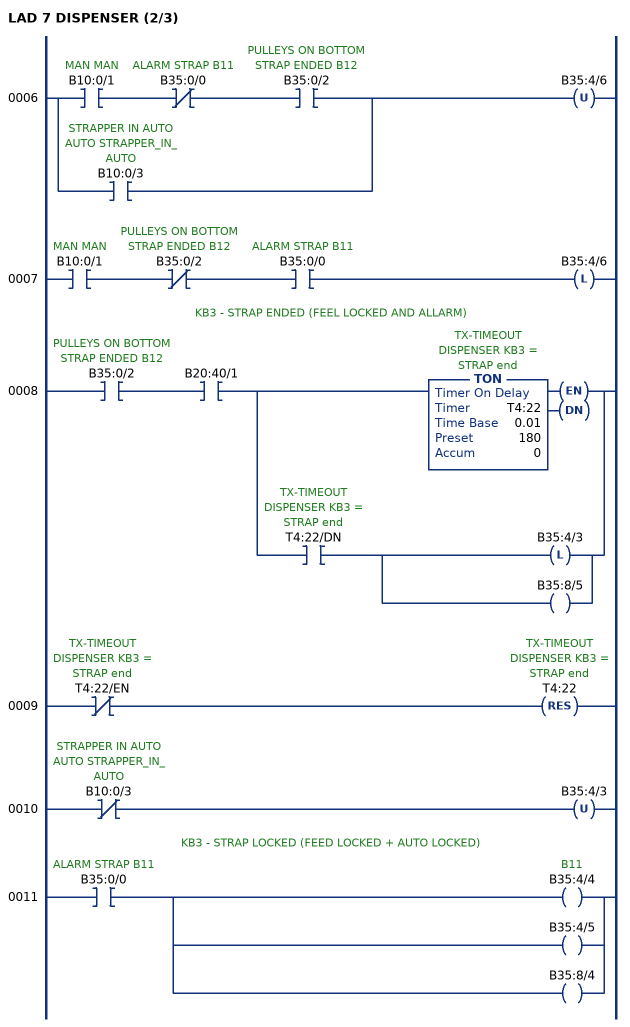
% Rung: 6 %
SOR BST XIC B10:0/1 XIO B35:0/0 XIC B35:0/2 NXB XIC B10:0/3 BND OTU B35:4/6 EOR
%   B10:0/1  MAN  "MAN" %
%   B35:0/0  B11  "ALARM STRAP" %
%   B35:0/2  B12  "PULLEYS ON BOTTOM STRAP ENDED" %
%   B10:0/3  STRAPPER_IN_AUTO  "STRAPPER IN AUTO AUTO" %
% Rung: 7 %
SOR XIC B10:0/1 XIO B35:0/2 XIC B35:0/0 OTL B35:4/6 EOR
%   B10:0/1  MAN  "MAN" %
%   B35:0/2  B12  "PULLEYS ON BOTTOM STRAP ENDED" %
%   B35:0/0  B11  "ALARM STRAP" %
% Rung: 8 %
% KB3 - STRAP ENDED (FEEL LOCKED AND ALLARM) %
SOR XIC B35:0/2 XIC B20:40/1 BST TON T4:22 0.01 180 0 NXB XIC T4:22/DN BST OTL B35:4/3 NXB OTE B35:8/5 BND BND EOR
%   B35:0/2  B12  "PULLEYS ON BOTTOM STRAP ENDED" %
%   T4:22  "TX-TIMEOUT DISPENSER KB3 = STRAP end" %
% Rung: 9 %
SOR XIO T4:22/EN RES T4:22 EOR
%   T4:22  "TX-TIMEOUT DISPENSER KB3 = STRAP end" %
% Rung: 10 %
SOR XIO B10:0/3 OTU B35:4/3 EOR
%   B10:0/3  STRAPPER_IN_AUTO  "STRAPPER IN AUTO AUTO" %
% Rung: 11 %
% KB3 - STRAP LOCKED (FEED LOCKED + AUTO LOCKED) %
SOR XIC B35:0/0 BST OTE B35:4/4 NXB BST OTE B35:4/5 NXB OTE B35:8/4 BND BND EOR
%   B35:0/0  B11  "ALARM STRAP" %
%   B35:4/4  "B11" %

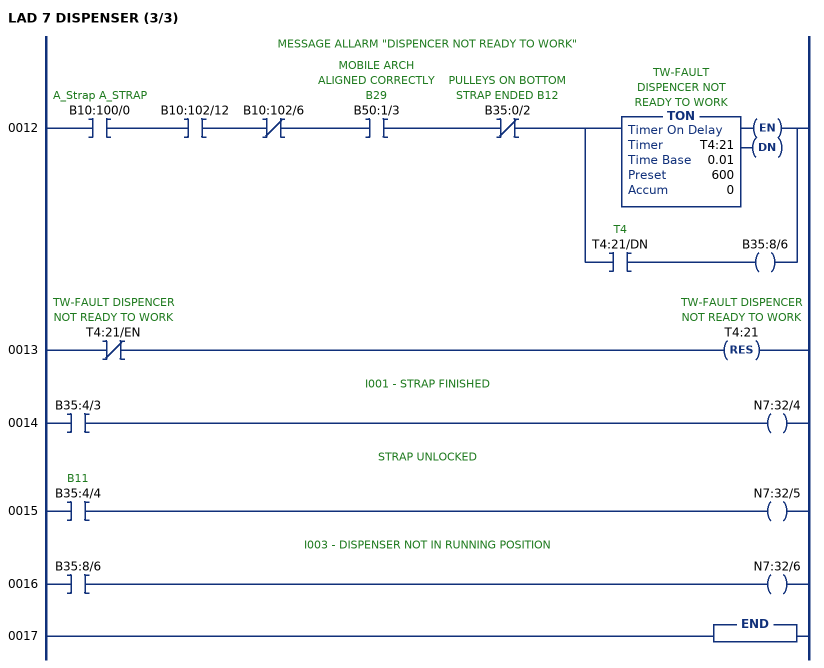
% Rung: 12 %
% MESSAGE ALLARM "DISPENCER NOT READY TO WORK" %
SOR XIC B10:100/0 XIC B10:102/12 XIO B10:102/6 XIC B50:1/3 XIO B35:0/2 BST TON T4:21 0.01 600 0 NXB XIC T4:21/DN OTE B35:8/6 BND EOR
%   B10:100/0  A_STRAP  "A_Strap" %
%   B50:1/3  B29  "MOBILE ARCH ALIGNED CORRECTLY" %
%   B35:0/2  B12  "PULLEYS ON BOTTOM STRAP ENDED" %
%   T4:21  "TW-FAULT DISPENCER NOT READY TO WORK" %
%   T4:21/DN  T4 %
% Rung: 13 %
SOR XIO T4:21/EN RES T4:21 EOR
%   T4:21  "TW-FAULT DISPENCER NOT READY TO WORK" %
% Rung: 14 %
% I001 - STRAP FINISHED %
SOR XIC B35:4/3 OTE N7:32/4 EOR
% Rung: 15 %
% STRAP UNLOCKED %
SOR XIC B35:4/4 OTE N7:32/5 EOR
%   B35:4/4  "B11" %
% Rung: 16 %
% I003 - DISPENSER NOT IN RUNNING POSITION %
SOR XIC B35:8/6 OTE N7:32/6 EOR
% Rung: 17 %
SOR END EOR

LADDER 8 "MH600"
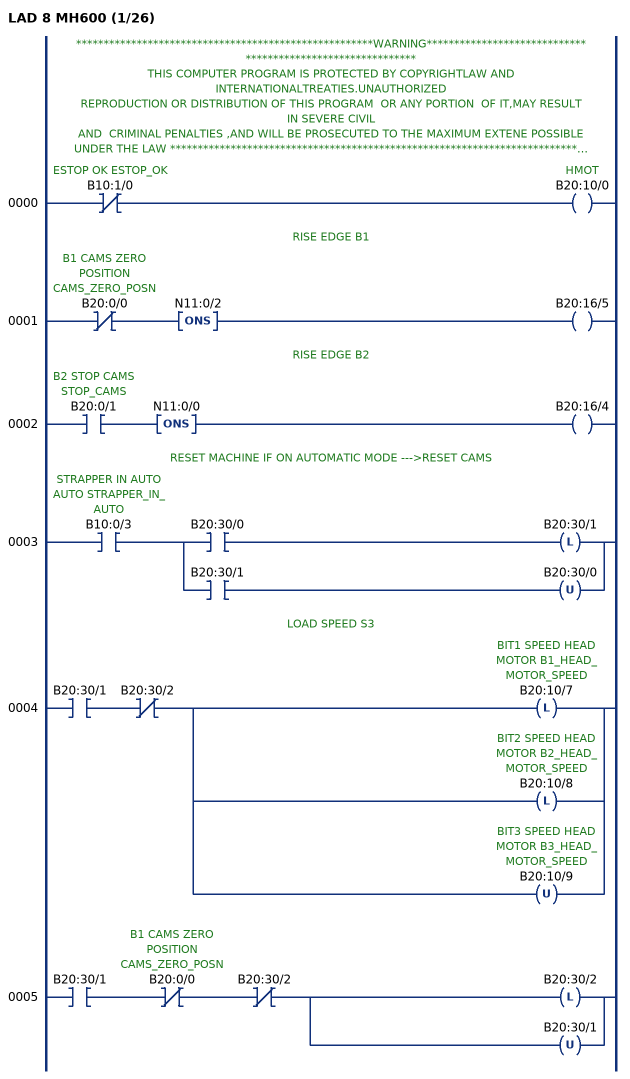
% Rung: 0 %
% ******************************************************WARNING************************************************************
% THIS COMPUTER PROGRAM IS PROTECTED BY COPYRIGHTLAW AND  INTERNATIONALTREATIES.UNAUTHORIZED
%  REPRODUCTION OR DISTRIBUTION OF THIS PROGRAM  OR ANY PORTION  OF IT,MAY RESULT IN SEVERE CIVIL
% AND  CRIMINAL PENALTIES ,AND WILL BE PROSECUTED TO THE MAXIMUM EXTENE POSSIBLE  UNDER THE LAW ************************************************************************************************************************** %
SOR XIO B10:1/0 OTE B20:10/0 EOR
%   B10:1/0  ESTOP_OK  "ESTOP OK" %
%   B20:10/0  "HMOT" %
% Rung: 1 %
% RISE EDGE B1 %
SOR XIO B20:0/0 ONS N11:0/2 OTE B20:16/5 EOR
%   B20:0/0  CAMS_ZERO_POSN  "B1 CAMS ZERO POSITION" %
% Rung: 2 %
% RISE EDGE B2 %
SOR XIC B20:0/1 ONS N11:0/0 OTE B20:16/4 EOR
%   B20:0/1  STOP_CAMS  "B2 STOP CAMS" %
% Rung: 3 %
% RESET MACHINE IF ON AUTOMATIC MODE --->RESET CAMS %
SOR XIC B10:0/3 BST XIC B20:30/0 OTL B20:30/1 NXB XIC B20:30/1 OTU B20:30/0 BND EOR
%   B10:0/3  STRAPPER_IN_AUTO  "STRAPPER IN AUTO AUTO" %
% Rung: 4 %
% LOAD SPEED S3 %
SOR XIC B20:30/1 XIO B20:30/2 BST OTL B20:10/7 NXB BST OTL B20:10/8 NXB OTU B20:10/9 BND BND EOR
%   B20:10/7  B1_HEAD_MOTOR_SPEED  "BIT1 SPEED HEAD MOTOR" %
%   B20:10/8  B2_HEAD_MOTOR_SPEED  "BIT2 SPEED HEAD MOTOR" %
%   B20:10/9  B3_HEAD_MOTOR_SPEED  "BIT3 SPEED HEAD MOTOR" %
% Rung: 5 %
SOR XIC B20:30/1 XIO B20:0/0 XIO B20:30/2 BST OTL B20:30/2 NXB OTU B20:30/1 BND EOR
%   B20:0/0  CAMS_ZERO_POSN  "B1 CAMS ZERO POSITION" %

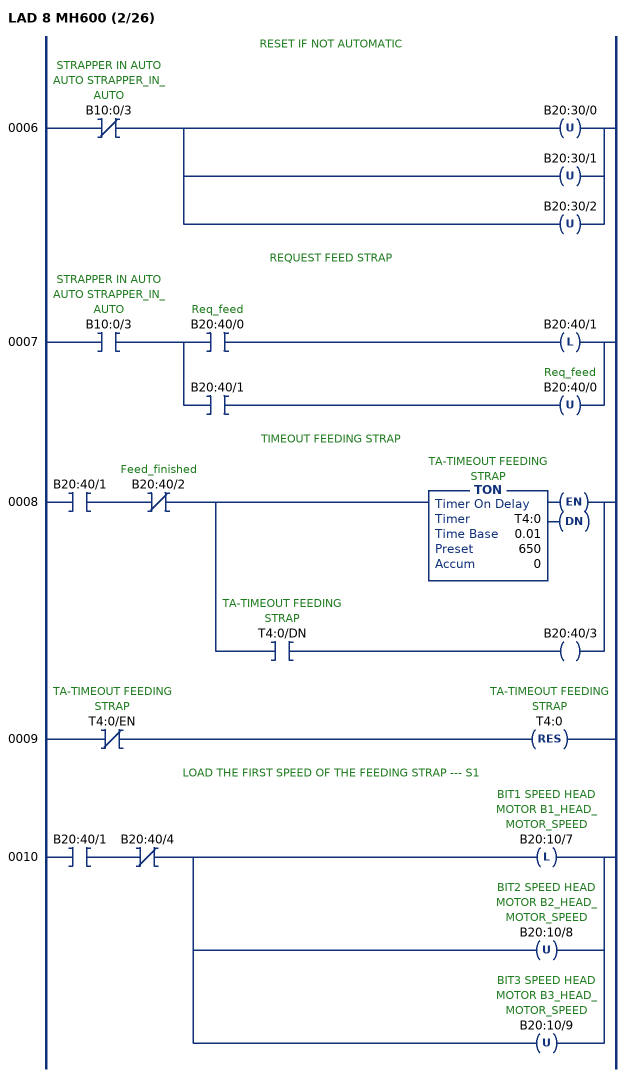
% Rung: 6 %
% RESET IF NOT AUTOMATIC %
SOR XIO B10:0/3 BST OTU B20:30/0 NXB BST OTU B20:30/1 NXB OTU B20:30/2 BND BND EOR
%   B10:0/3  STRAPPER_IN_AUTO  "STRAPPER IN AUTO AUTO" %
% Rung: 7 %
% REQUEST FEED STRAP %
SOR XIC B10:0/3 BST XIC B20:40/0 OTL B20:40/1 NXB XIC B20:40/1 OTU B20:40/0 BND EOR
%   B10:0/3  STRAPPER_IN_AUTO  "STRAPPER IN AUTO AUTO" %
%   B20:40/0  "Req_feed" %
% Rung: 8 %
% TIMEOUT FEEDING STRAP %
SOR XIC B20:40/1 XIO B20:40/2 BST TON T4:0 0.01 650 0 NXB XIC T4:0/DN OTE B20:40/3 BND EOR
%   B20:40/2  "Feed_finished" %
%   T4:0  "TA-TIMEOUT FEEDING STRAP" %
% Rung: 9 %
SOR XIO T4:0/EN RES T4:0 EOR
%   T4:0  "TA-TIMEOUT FEEDING STRAP" %
% Rung: 10 %
% LOAD THE FIRST SPEED OF THE FEEDING STRAP --- S1 %
SOR XIC B20:40/1 XIO B20:40/4 BST OTL B20:10/7 NXB BST OTU B20:10/8 NXB OTU B20:10/9 BND BND EOR
%   B20:10/7  B1_HEAD_MOTOR_SPEED  "BIT1 SPEED HEAD MOTOR" %
%   B20:10/8  B2_HEAD_MOTOR_SPEED  "BIT2 SPEED HEAD MOTOR" %
%   B20:10/9  B3_HEAD_MOTOR_SPEED  "BIT3 SPEED HEAD MOTOR" %

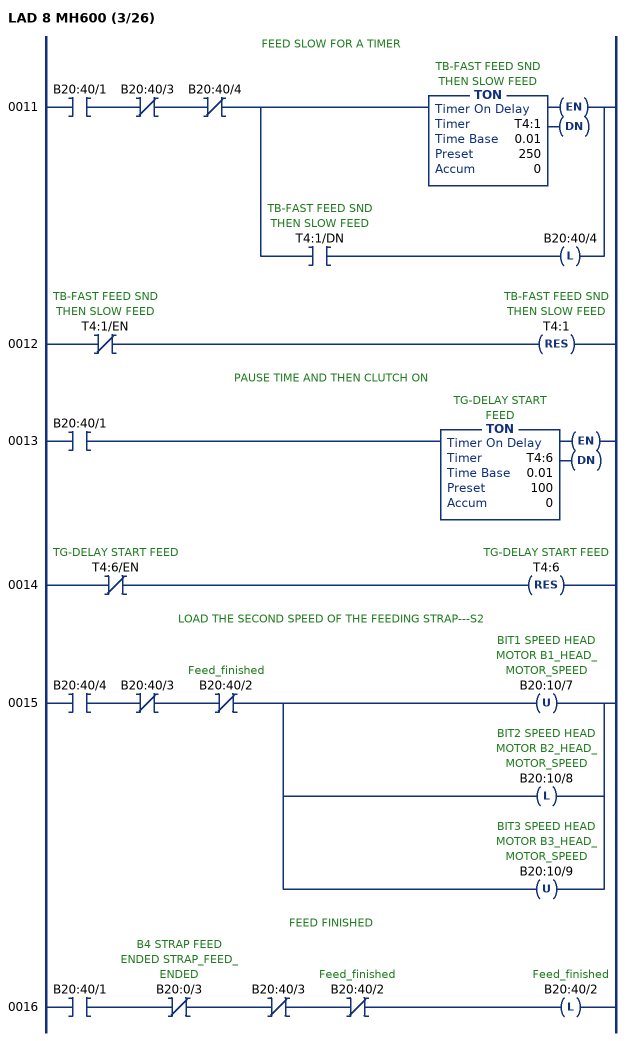
% Rung: 11 %
% FEED SLOW FOR A TIMER %
SOR XIC B20:40/1 XIO B20:40/3 XIO B20:40/4 BST TON T4:1 0.01 250 0 NXB XIC T4:1/DN OTL B20:40/4 BND EOR
%   T4:1  "TB-FAST FEED SND THEN SLOW FEED" %
% Rung: 12 %
SOR XIO T4:1/EN RES T4:1 EOR
%   T4:1  "TB-FAST FEED SND THEN SLOW FEED" %
% Rung: 13 %
% PAUSE TIME AND THEN CLUTCH ON %
SOR XIC B20:40/1 TON T4:6 0.01 100 0 EOR
%   T4:6  "TG-DELAY START FEED" %
% Rung: 14 %
SOR XIO T4:6/EN RES T4:6 EOR
%   T4:6  "TG-DELAY START FEED" %
% Rung: 15 %
% LOAD THE SECOND SPEED OF THE FEEDING STRAP---S2 %
SOR XIC B20:40/4 XIO B20:40/3 XIO B20:40/2 BST OTU B20:10/7 NXB BST OTL B20:10/8 NXB OTU B20:10/9 BND BND EOR
%   B20:40/2  "Feed_finished" %
%   B20:10/7  B1_HEAD_MOTOR_SPEED  "BIT1 SPEED HEAD MOTOR" %
%   B20:10/8  B2_HEAD_MOTOR_SPEED  "BIT2 SPEED HEAD MOTOR" %
%   B20:10/9  B3_HEAD_MOTOR_SPEED  "BIT3 SPEED HEAD MOTOR" %
% Rung: 16 %
% FEED FINISHED %
SOR XIC B20:40/1 XIO B20:0/3 XIO B20:40/3 XIO B20:40/2 OTL B20:40/2 EOR
%   B20:0/3  STRAP_FEED_ENDED  "B4 STRAP FEED ENDED" %
%   B20:40/2  "Feed_finished" %

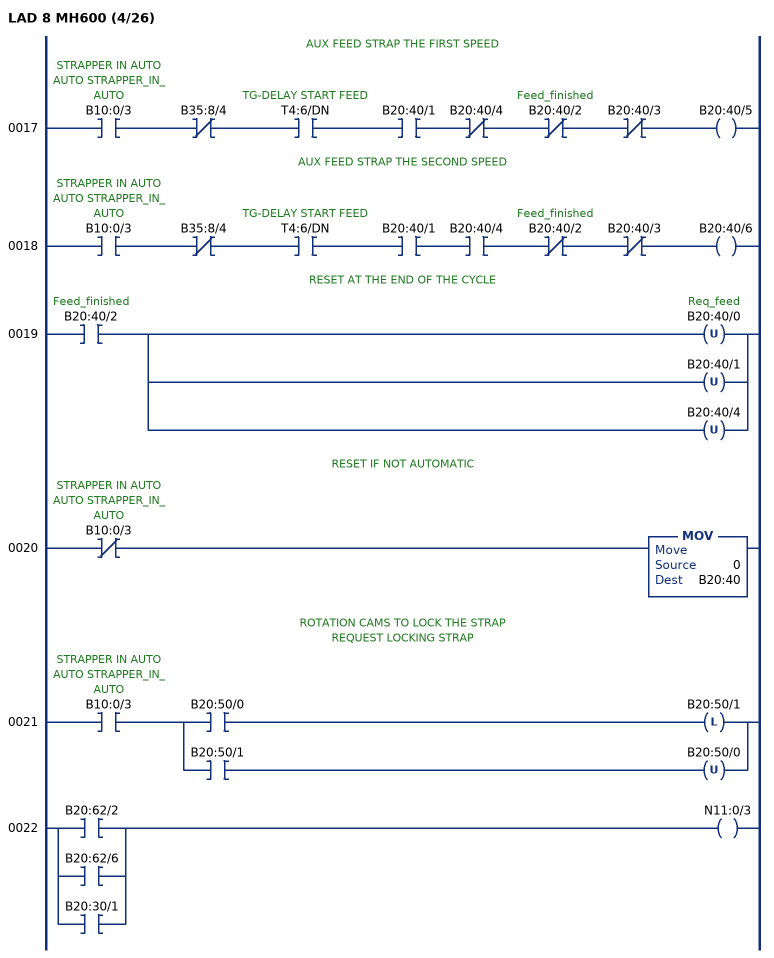
% Rung: 17 %
% AUX FEED STRAP THE FIRST SPEED %
SOR XIC B10:0/3 XIO B35:8/4 XIC T4:6/DN XIC B20:40/1 XIO B20:40/4 XIO B20:40/2 XIO B20:40/3 OTE B20:40/5 EOR
%   B10:0/3  STRAPPER_IN_AUTO  "STRAPPER IN AUTO AUTO" %
%   T4:6  "TG-DELAY START FEED" %
%   B20:40/2  "Feed_finished" %
% Rung: 18 %
% AUX FEED STRAP THE SECOND SPEED %
SOR XIC B10:0/3 XIO B35:8/4 XIC T4:6/DN XIC B20:40/1 XIC B20:40/4 XIO B20:40/2 XIO B20:40/3 OTE B20:40/6 EOR
%   B10:0/3  STRAPPER_IN_AUTO  "STRAPPER IN AUTO AUTO" %
%   T4:6  "TG-DELAY START FEED" %
%   B20:40/2  "Feed_finished" %
% Rung: 19 %
% RESET AT THE END OF THE CYCLE %
SOR XIC B20:40/2 BST OTU B20:40/0 NXB BST OTU B20:40/1 NXB OTU B20:40/4 BND BND EOR
%   B20:40/2  "Feed_finished" %
%   B20:40/0  "Req_feed" %
% Rung: 20 %
% RESET IF NOT AUTOMATIC %
SOR XIO B10:0/3 MOV 0 B20:40 EOR
%   B10:0/3  STRAPPER_IN_AUTO  "STRAPPER IN AUTO AUTO" %
% Rung: 21 %
% ROTATION CAMS TO LOCK THE STRAP
% REQUEST LOCKING STRAP %
SOR XIC B10:0/3 BST XIC B20:50/0 OTL B20:50/1 NXB XIC B20:50/1 OTU B20:50/0 BND EOR
%   B10:0/3  STRAPPER_IN_AUTO  "STRAPPER IN AUTO AUTO" %
% Rung: 22 %
SOR BST XIC B20:62/2 NXB BST XIC B20:62/6 NXB XIC B20:30/1 BND BND OTE N11:0/3 EOR

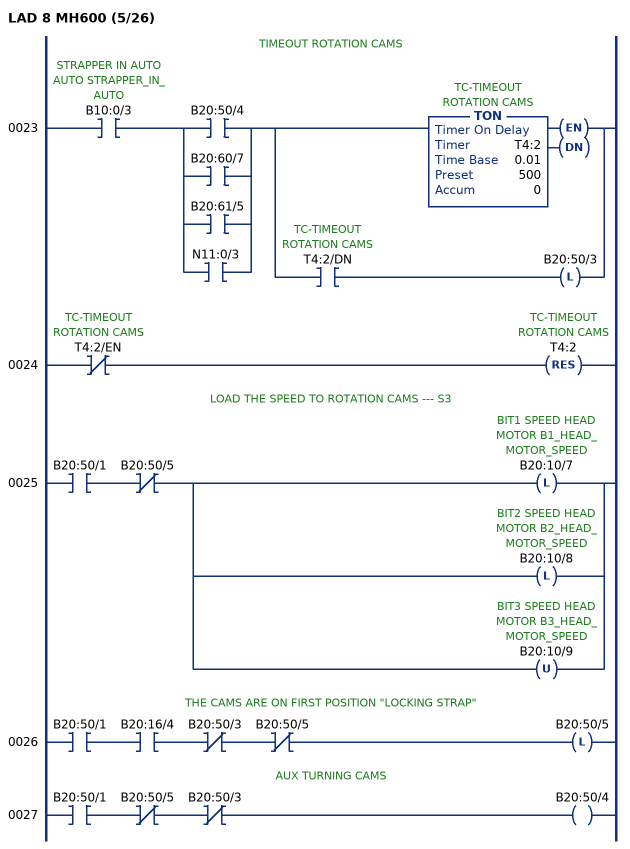
% Rung: 23 %
% TIMEOUT ROTATION CAMS %
SOR XIC B10:0/3 BST XIC B20:50/4 NXB BST XIC B20:60/7 NXB BST XIC B20:61/5 NXB XIC N11:0/3 BND BND BND BST TON T4:2 0.01 500 0 NXB XIC T4:2/DN OTL B20:50/3 BND EOR
%   B10:0/3  STRAPPER_IN_AUTO  "STRAPPER IN AUTO AUTO" %
%   T4:2  "TC-TIMEOUT ROTATION CAMS" %
% Rung: 24 %
SOR XIO T4:2/EN RES T4:2 EOR
%   T4:2  "TC-TIMEOUT ROTATION CAMS" %
% Rung: 25 %
% LOAD THE SPEED TO ROTATION CAMS --- S3 %
SOR XIC B20:50/1 XIO B20:50/5 BST OTL B20:10/7 NXB BST OTL B20:10/8 NXB OTU B20:10/9 BND BND EOR
%   B20:10/7  B1_HEAD_MOTOR_SPEED  "BIT1 SPEED HEAD MOTOR" %
%   B20:10/8  B2_HEAD_MOTOR_SPEED  "BIT2 SPEED HEAD MOTOR" %
%   B20:10/9  B3_HEAD_MOTOR_SPEED  "BIT3 SPEED HEAD MOTOR" %
% Rung: 26 %
% THE CAMS ARE ON FIRST POSITION "LOCKING STRAP" %
SOR XIC B20:50/1 XIC B20:16/4 XIO B20:50/3 XIO B20:50/5 OTL B20:50/5 EOR
% Rung: 27 %
% AUX TURNING CAMS %
SOR XIC B20:50/1 XIO B20:50/5 XIO B20:50/3 OTE B20:50/4 EOR

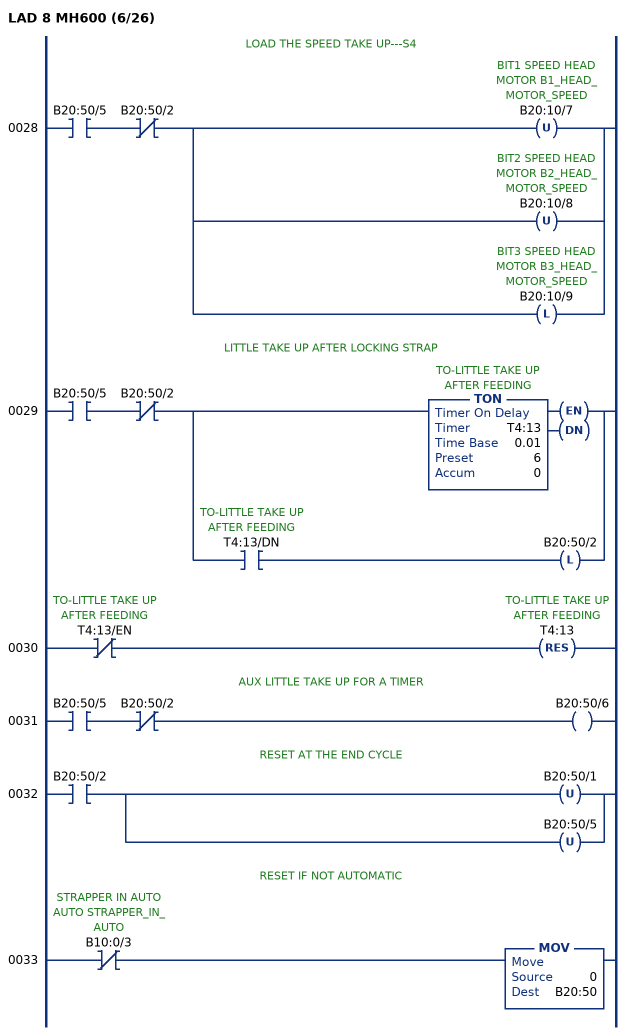
% Rung: 28 %
% LOAD THE SPEED TAKE UP---S4 %
SOR XIC B20:50/5 XIO B20:50/2 BST OTU B20:10/7 NXB BST OTU B20:10/8 NXB OTL B20:10/9 BND BND EOR
%   B20:10/7  B1_HEAD_MOTOR_SPEED  "BIT1 SPEED HEAD MOTOR" %
%   B20:10/8  B2_HEAD_MOTOR_SPEED  "BIT2 SPEED HEAD MOTOR" %
%   B20:10/9  B3_HEAD_MOTOR_SPEED  "BIT3 SPEED HEAD MOTOR" %
% Rung: 29 %
% LITTLE TAKE UP AFTER LOCKING STRAP %
SOR XIC B20:50/5 XIO B20:50/2 BST TON T4:13 0.01 6 0 NXB XIC T4:13/DN OTL B20:50/2 BND EOR
%   T4:13  "TO-LITTLE TAKE UP AFTER FEEDING" %
% Rung: 30 %
SOR XIO T4:13/EN RES T4:13 EOR
%   T4:13  "TO-LITTLE TAKE UP AFTER FEEDING" %
% Rung: 31 %
% AUX LITTLE TAKE UP FOR A TIMER %
SOR XIC B20:50/5 XIO B20:50/2 OTE B20:50/6 EOR
% Rung: 32 %
% RESET AT THE END CYCLE %
SOR XIC B20:50/2 BST OTU B20:50/1 NXB OTU B20:50/5 BND EOR
% Rung: 33 %
% RESET IF NOT AUTOMATIC %
SOR XIO B10:0/3 MOV 0 B20:50 EOR
%   B10:0/3  STRAPPER_IN_AUTO  "STRAPPER IN AUTO AUTO" %

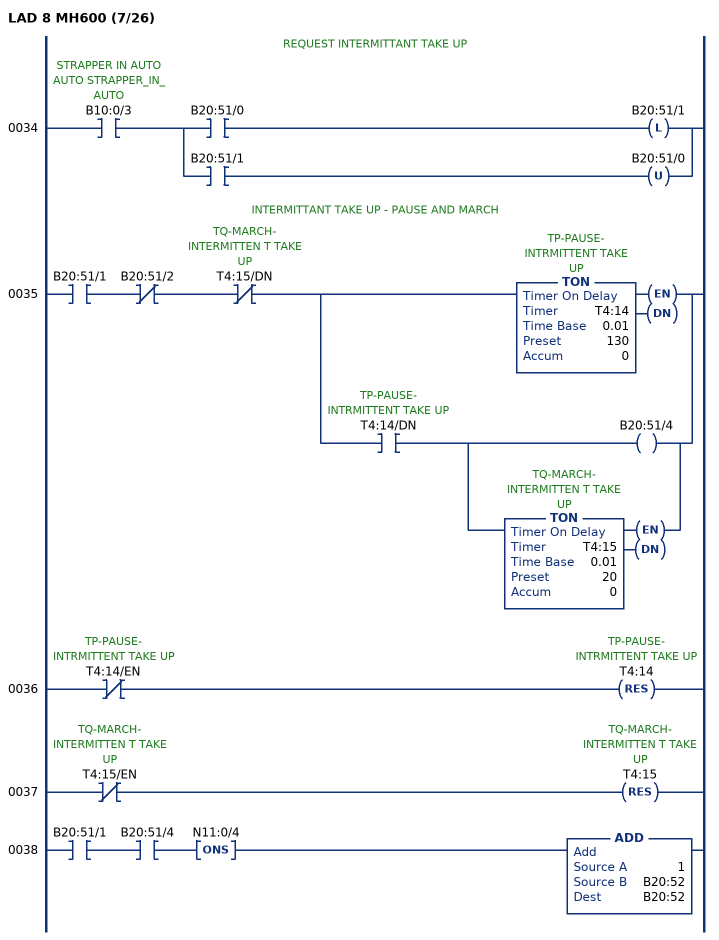
% Rung: 34 %
% REQUEST INTERMITTANT TAKE UP %
SOR XIC B10:0/3 BST XIC B20:51/0 OTL B20:51/1 NXB XIC B20:51/1 OTU B20:51/0 BND EOR
%   B10:0/3  STRAPPER_IN_AUTO  "STRAPPER IN AUTO AUTO" %
% Rung: 35 %
% INTERMITTANT TAKE UP - PAUSE AND MARCH %
SOR XIC B20:51/1 XIO B20:51/2 XIO T4:15/DN BST TON T4:14 0.01 130 0 NXB XIC T4:14/DN BST OTE B20:51/4 NXB TON T4:15 0.01 20 0 BND BND EOR
%   T4:15  "TQ-MARCH-INTERMITTEN T TAKE UP" %
%   T4:14  "TP-PAUSE-INTRMITTENT TAKE UP" %
% Rung: 36 %
SOR XIO T4:14/EN RES T4:14 EOR
%   T4:14  "TP-PAUSE-INTRMITTENT TAKE UP" %
% Rung: 37 %
SOR XIO T4:15/EN RES T4:15 EOR
%   T4:15  "TQ-MARCH-INTERMITTEN T TAKE UP" %
% Rung: 38 %
SOR XIC B20:51/1 XIC B20:51/4 ONS N11:0/4 ADD 1 B20:52 B20:52 EOR

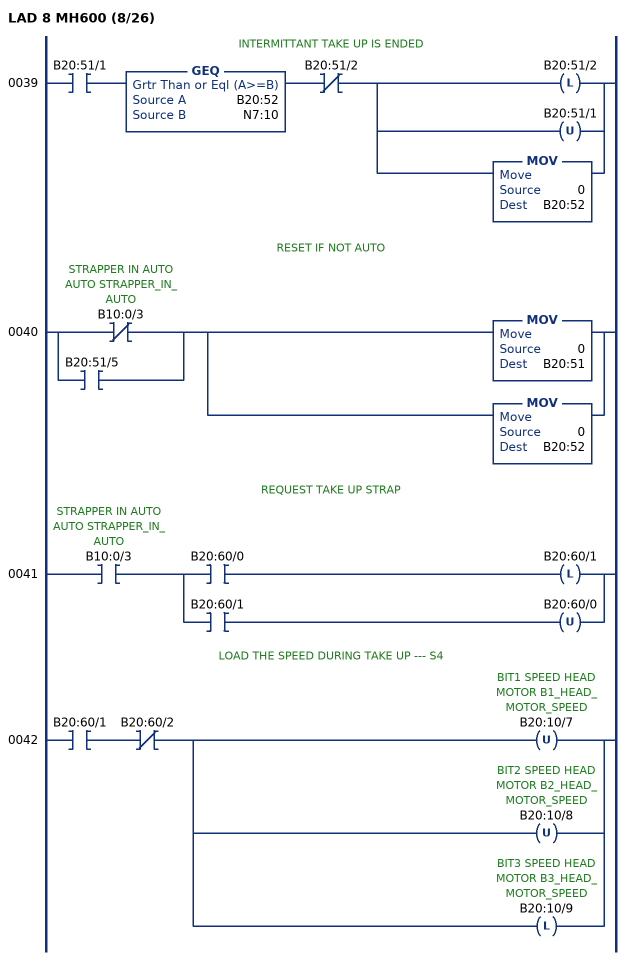
% Rung: 39 %
% INTERMITTANT TAKE UP IS ENDED %
SOR XIC B20:51/1 GEQ B20:52 N7:10 XIO B20:51/2 BST OTL B20:51/2 NXB BST OTU B20:51/1 NXB MOV 0 B20:52 BND BND EOR
%   N7:10  "NUMBER OF SHOOTS INTERMITTANT TAKE UP" %
% Rung: 40 %
% RESET IF NOT AUTO %
SOR BST XIO B10:0/3 NXB XIC B20:51/5 BND BST MOV 0 B20:51 NXB MOV 0 B20:52 BND EOR
%   B10:0/3  STRAPPER_IN_AUTO  "STRAPPER IN AUTO AUTO" %
% Rung: 41 %
% REQUEST TAKE UP STRAP %
SOR XIC B10:0/3 BST XIC B20:60/0 OTL B20:60/1 NXB XIC B20:60/1 OTU B20:60/0 BND EOR
%   B10:0/3  STRAPPER_IN_AUTO  "STRAPPER IN AUTO AUTO" %
% Rung: 42 %
% LOAD THE SPEED DURING TAKE UP --- S4 %
SOR XIC B20:60/1 XIO B20:60/2 BST OTU B20:10/7 NXB BST OTU B20:10/8 NXB OTL B20:10/9 BND BND EOR
%   B20:10/7  B1_HEAD_MOTOR_SPEED  "BIT1 SPEED HEAD MOTOR" %
%   B20:10/8  B2_HEAD_MOTOR_SPEED  "BIT2 SPEED HEAD MOTOR" %
%   B20:10/9  B3_HEAD_MOTOR_SPEED  "BIT3 SPEED HEAD MOTOR" %

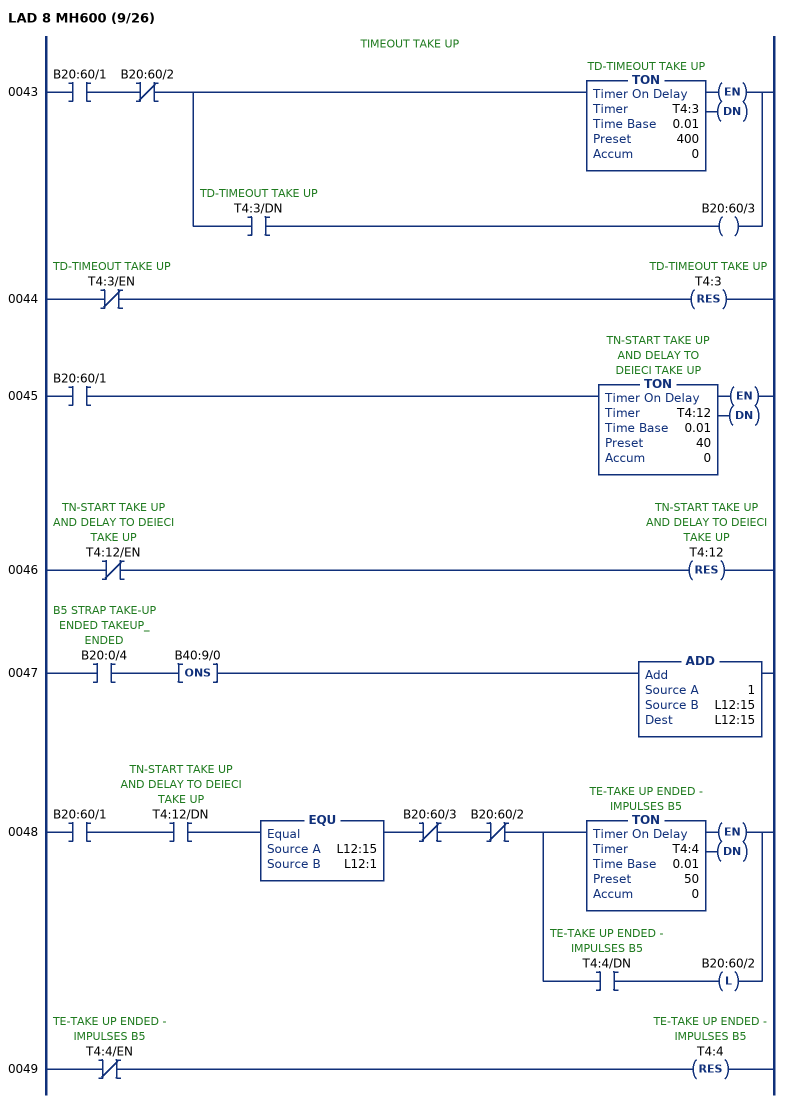
% Rung: 43 %
% TIMEOUT TAKE UP %
SOR XIC B20:60/1 XIO B20:60/2 BST TON T4:3 0.01 400 0 NXB XIC T4:3/DN OTE B20:60/3 BND EOR
%   T4:3  "TD-TIMEOUT TAKE UP" %
% Rung: 44 %
SOR XIO T4:3/EN RES T4:3 EOR
%   T4:3  "TD-TIMEOUT TAKE UP" %
% Rung: 45 %
SOR XIC B20:60/1 TON T4:12 0.01 40 0 EOR
%   T4:12  "TN-START TAKE UP AND DELAY TO DEIECI TAKE UP" %
% Rung: 46 %
SOR XIO T4:12/EN RES T4:12 EOR
%   T4:12  "TN-START TAKE UP AND DELAY TO DEIECI TAKE UP" %
% Rung: 47 %
SOR XIC B20:0/4 ONS B40:9/0 ADD 1 L12:15 L12:15 EOR
%   B20:0/4  TAKEUP_ENDED  "B5 STRAP TAKE-UP ENDED" %
% Rung: 48 %
SOR XIC B20:60/1 XIC T4:12/DN EQU L12:15 L12:1 XIO B20:60/3 XIO B20:60/2 BST TON T4:4 0.01 50 0 NXB XIC T4:4/DN OTL B20:60/2 BND EOR
%   T4:12  "TN-START TAKE UP AND DELAY TO DEIECI TAKE UP" %
%   T4:4  "TE-TAKE UP ENDED - IMPULSES B5" %
% Rung: 49 %
SOR XIO T4:4/EN RES T4:4 EOR
%   T4:4  "TE-TAKE UP ENDED - IMPULSES B5" %

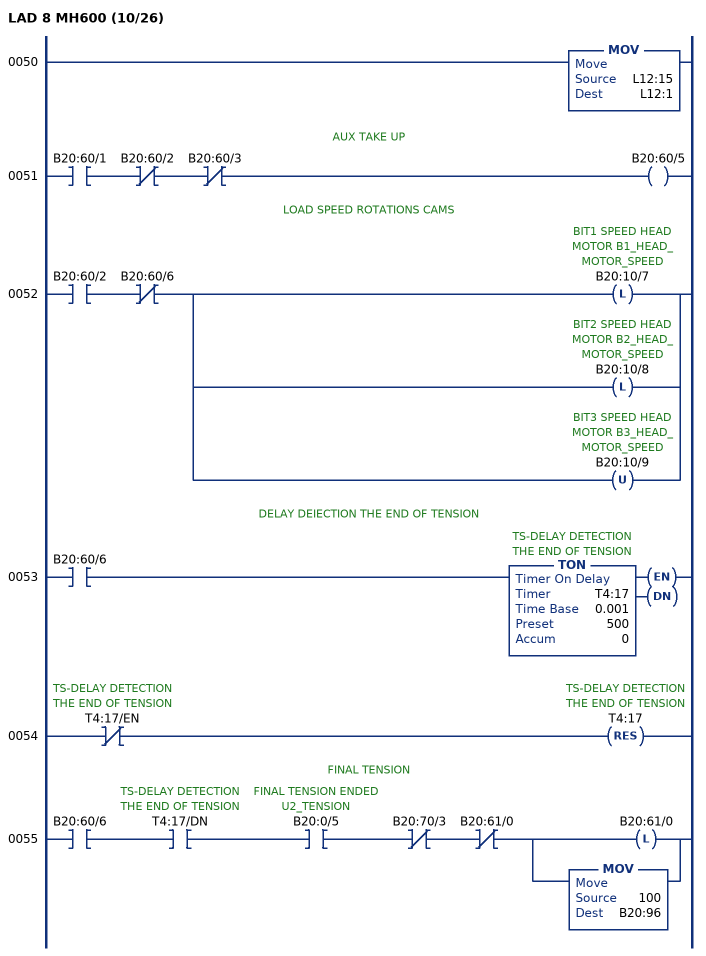
% Rung: 50 %
SOR MOV L12:15 L12:1 EOR
% Rung: 51 %
% AUX TAKE UP %
SOR XIC B20:60/1 XIO B20:60/2 XIO B20:60/3 OTE B20:60/5 EOR
% Rung: 52 %
% LOAD SPEED ROTATIONS CAMS %
SOR XIC B20:60/2 XIO B20:60/6 BST OTL B20:10/7 NXB BST OTL B20:10/8 NXB OTU B20:10/9 BND BND EOR
%   B20:10/7  B1_HEAD_MOTOR_SPEED  "BIT1 SPEED HEAD MOTOR" %
%   B20:10/8  B2_HEAD_MOTOR_SPEED  "BIT2 SPEED HEAD MOTOR" %
%   B20:10/9  B3_HEAD_MOTOR_SPEED  "BIT3 SPEED HEAD MOTOR" %
% Rung: 53 %
% DELAY DEIECTION THE END OF TENSION %
SOR XIC B20:60/6 TON T4:17 0.001 500 0 EOR
%   T4:17  "TS-DELAY DETECTION THE END OF TENSION" %
% Rung: 54 %
SOR XIO T4:17/EN RES T4:17 EOR
%   T4:17  "TS-DELAY DETECTION THE END OF TENSION" %
% Rung: 55 %
% FINAL TENSION %
SOR XIC B20:60/6 XIC T4:17/DN XIC B20:0/5 XIO B20:70/3 XIO B20:61/0 BST OTL B20:61/0 NXB MOV 100 B20:96 BND EOR
%   T4:17  "TS-DELAY DETECTION THE END OF TENSION" %
%   B20:0/5  U2_TENSION  "FINAL TENSION ENDED" %

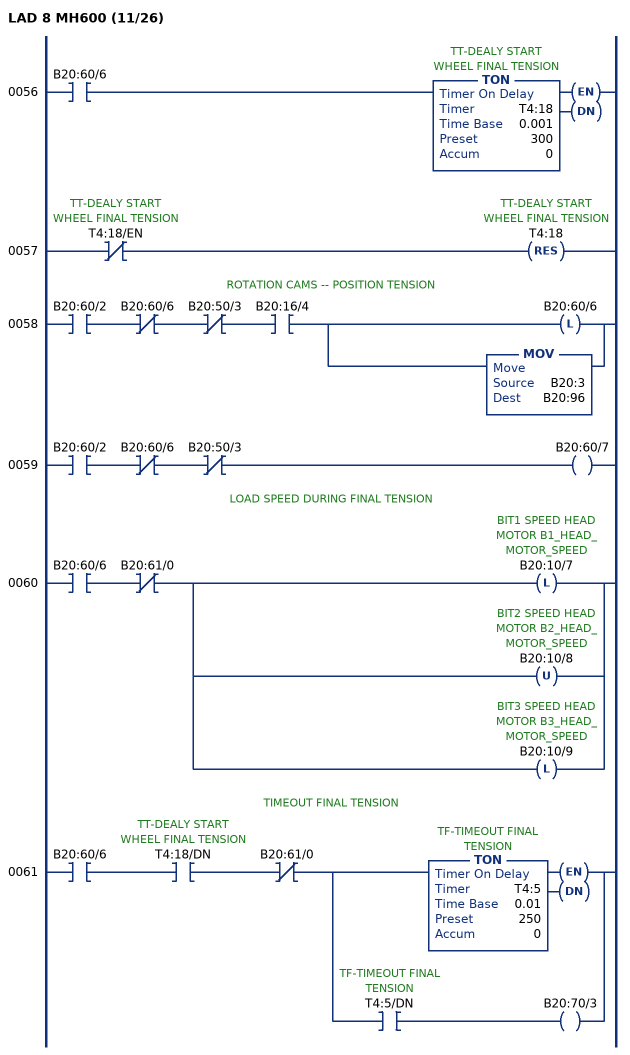
% Rung: 56 %
SOR XIC B20:60/6 TON T4:18 0.001 300 0 EOR
%   T4:18  "TT-DEALY START WHEEL FINAL TENSION" %
% Rung: 57 %
SOR XIO T4:18/EN RES T4:18 EOR
%   T4:18  "TT-DEALY START WHEEL FINAL TENSION" %
% Rung: 58 %
% ROTATION CAMS -- POSITION TENSION %
SOR XIC B20:60/2 XIO B20:60/6 XIO B20:50/3 XIC B20:16/4 BST OTL B20:60/6 NXB MOV B20:3 B20:96 BND EOR
% Rung: 59 %
SOR XIC B20:60/2 XIO B20:60/6 XIO B20:50/3 OTE B20:60/7 EOR
% Rung: 60 %
% LOAD SPEED DURING FINAL TENSION %
SOR XIC B20:60/6 XIO B20:61/0 BST OTL B20:10/7 NXB BST OTU B20:10/8 NXB OTL B20:10/9 BND BND EOR
%   B20:10/7  B1_HEAD_MOTOR_SPEED  "BIT1 SPEED HEAD MOTOR" %
%   B20:10/8  B2_HEAD_MOTOR_SPEED  "BIT2 SPEED HEAD MOTOR" %
%   B20:10/9  B3_HEAD_MOTOR_SPEED  "BIT3 SPEED HEAD MOTOR" %
% Rung: 61 %
% TIMEOUT FINAL TENSION %
SOR XIC B20:60/6 XIC T4:18/DN XIO B20:61/0 BST TON T4:5 0.01 250 0 NXB XIC T4:5/DN OTE B20:70/3 BND EOR
%   T4:18  "TT-DEALY START WHEEL FINAL TENSION" %
%   T4:5  "TF-TIMEOUT FINAL TENSION" %

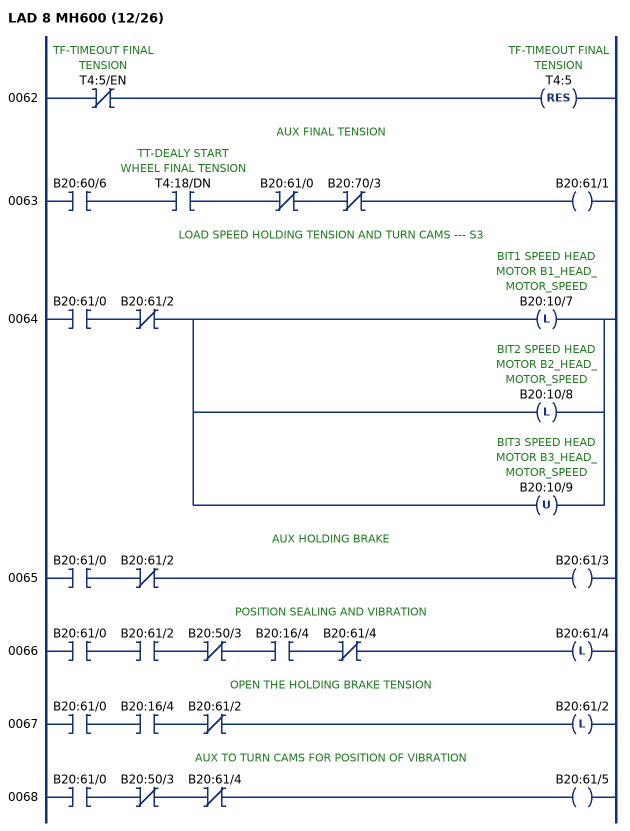
% Rung: 62 %
SOR XIO T4:5/EN RES T4:5 EOR
%   T4:5  "TF-TIMEOUT FINAL TENSION" %
% Rung: 63 %
% AUX FINAL TENSION %
SOR XIC B20:60/6 XIC T4:18/DN XIO B20:61/0 XIO B20:70/3 OTE B20:61/1 EOR
%   T4:18  "TT-DEALY START WHEEL FINAL TENSION" %
% Rung: 64 %
% LOAD SPEED HOLDING TENSION AND TURN CAMS --- S3 %
SOR XIC B20:61/0 XIO B20:61/2 BST OTL B20:10/7 NXB BST OTL B20:10/8 NXB OTU B20:10/9 BND BND EOR
%   B20:10/7  B1_HEAD_MOTOR_SPEED  "BIT1 SPEED HEAD MOTOR" %
%   B20:10/8  B2_HEAD_MOTOR_SPEED  "BIT2 SPEED HEAD MOTOR" %
%   B20:10/9  B3_HEAD_MOTOR_SPEED  "BIT3 SPEED HEAD MOTOR" %
% Rung: 65 %
% AUX HOLDING BRAKE %
SOR XIC B20:61/0 XIO B20:61/2 OTE B20:61/3 EOR
% Rung: 66 %
% POSITION SEALING AND VIBRATION %
SOR XIC B20:61/0 XIC B20:61/2 XIO B20:50/3 XIC B20:16/4 XIO B20:61/4 OTL B20:61/4 EOR
% Rung: 67 %
% OPEN THE HOLDING BRAKE TENSION %
SOR XIC B20:61/0 XIC B20:16/4 XIO B20:61/2 OTL B20:61/2 EOR
% Rung: 68 %
% AUX TO TURN CAMS FOR POSITION OF VIBRATION %
SOR XIC B20:61/0 XIO B20:50/3 XIO B20:61/4 OTE B20:61/5 EOR

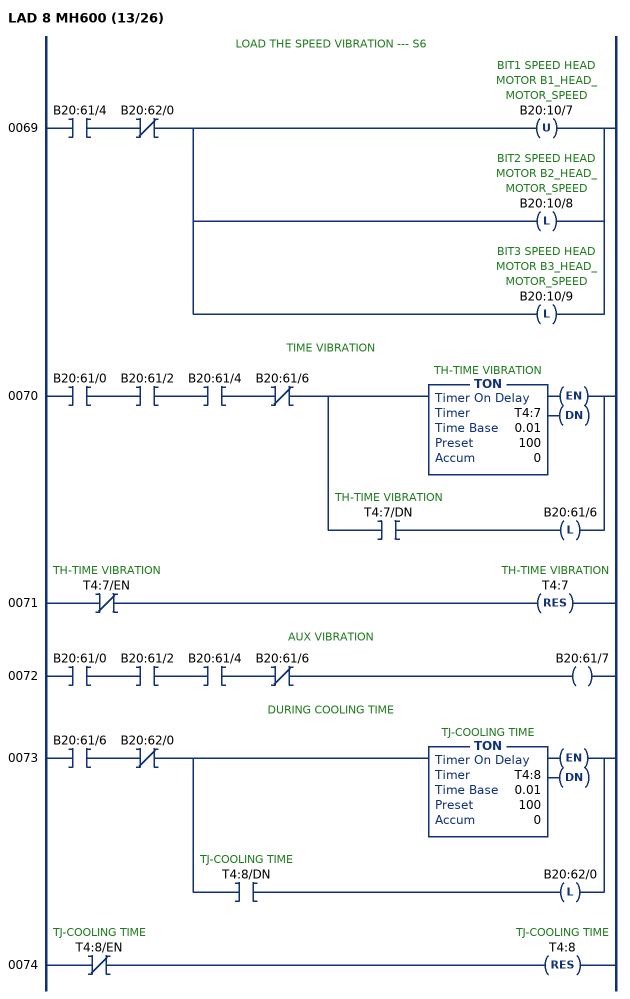
% Rung: 69 %
% LOAD THE SPEED VIBRATION --- S6 %
SOR XIC B20:61/4 XIO B20:62/0 BST OTU B20:10/7 NXB BST OTL B20:10/8 NXB OTL B20:10/9 BND BND EOR
%   B20:10/7  B1_HEAD_MOTOR_SPEED  "BIT1 SPEED HEAD MOTOR" %
%   B20:10/8  B2_HEAD_MOTOR_SPEED  "BIT2 SPEED HEAD MOTOR" %
%   B20:10/9  B3_HEAD_MOTOR_SPEED  "BIT3 SPEED HEAD MOTOR" %
% Rung: 70 %
% TIME VIBRATION %
SOR XIC B20:61/0 XIC B20:61/2 XIC B20:61/4 XIO B20:61/6 BST TON T4:7 0.01 100 0 NXB XIC T4:7/DN OTL B20:61/6 BND EOR
%   T4:7  "TH-TIME VIBRATION" %
% Rung: 71 %
SOR XIO T4:7/EN RES T4:7 EOR
%   T4:7  "TH-TIME VIBRATION" %
% Rung: 72 %
% AUX VIBRATION %
SOR XIC B20:61/0 XIC B20:61/2 XIC B20:61/4 XIO B20:61/6 OTE B20:61/7 EOR
% Rung: 73 %
% DURING COOLING TIME %
SOR XIC B20:61/6 XIO B20:62/0 BST TON T4:8 0.01 100 0 NXB XIC T4:8/DN OTL B20:62/0 BND EOR
%   T4:8  "TJ-COOLING TIME" %
% Rung: 74 %
SOR XIO T4:8/EN RES T4:8 EOR
%   T4:8  "TJ-COOLING TIME" %

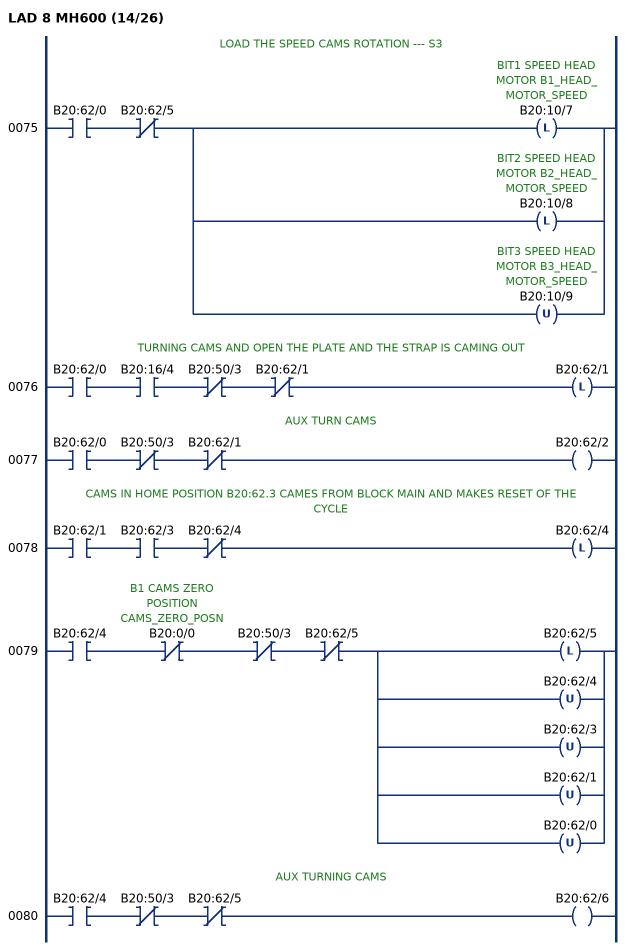
% Rung: 75 %
% LOAD THE SPEED CAMS ROTATION --- S3 %
SOR XIC B20:62/0 XIO B20:62/5 BST OTL B20:10/7 NXB BST OTL B20:10/8 NXB OTU B20:10/9 BND BND EOR
%   B20:10/7  B1_HEAD_MOTOR_SPEED  "BIT1 SPEED HEAD MOTOR" %
%   B20:10/8  B2_HEAD_MOTOR_SPEED  "BIT2 SPEED HEAD MOTOR" %
%   B20:10/9  B3_HEAD_MOTOR_SPEED  "BIT3 SPEED HEAD MOTOR" %
% Rung: 76 %
% TURNING CAMS AND OPEN THE PLATE AND THE STRAP IS CAMING OUT %
SOR XIC B20:62/0 XIC B20:16/4 XIO B20:50/3 XIO B20:62/1 OTL B20:62/1 EOR
% Rung: 77 %
% AUX TURN CAMS %
SOR XIC B20:62/0 XIO B20:50/3 XIO B20:62/1 OTE B20:62/2 EOR
% Rung: 78 %
% CAMS IN HOME POSITION B20:62.3 CAMES FROM BLOCK MAIN AND MAKES RESET OF THE CYCLE %
SOR XIC B20:62/1 XIC B20:62/3 XIO B20:62/4 OTL B20:62/4 EOR
% Rung: 79 %
SOR XIC B20:62/4 XIO B20:0/0 XIO B20:50/3 XIO B20:62/5 BST OTL B20:62/5 NXB BST OTU B20:62/4 NXB BST OTU B20:62/3 NXB BST OTU B20:62/1 NXB OTU B20:62/0 BND BND BND BND EOR
%   B20:0/0  CAMS_ZERO_POSN  "B1 CAMS ZERO POSITION" %
% Rung: 80 %
% AUX TURNING CAMS %
SOR XIC B20:62/4 XIO B20:50/3 XIO B20:62/5 OTE B20:62/6 EOR

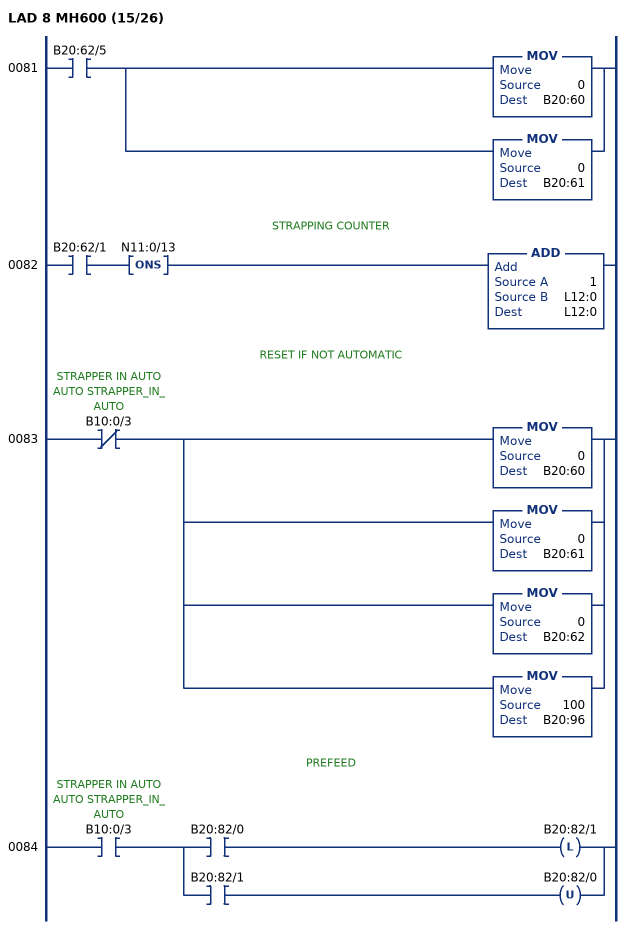
% Rung: 81 %
SOR XIC B20:62/5 BST MOV 0 B20:60 NXB MOV 0 B20:61 BND EOR
% Rung: 82 %
% STRAPPING COUNTER %
SOR XIC B20:62/1 ONS N11:0/13 ADD 1 L12:0 L12:0 EOR
% Rung: 83 %
% RESET IF NOT AUTOMATIC %
SOR XIO B10:0/3 BST BST MOV 0 B20:60 NXB MOV 0 B20:61 BND NXB BST MOV 0 B20:62 NXB MOV 100 B20:96 BND BND EOR
%   B10:0/3  STRAPPER_IN_AUTO  "STRAPPER IN AUTO AUTO" %
% Rung: 84 %
% PREFEED %
SOR XIC B10:0/3 BST XIC B20:82/0 OTL B20:82/1 NXB XIC B20:82/1 OTU B20:82/0 BND EOR
%   B10:0/3  STRAPPER_IN_AUTO  "STRAPPER IN AUTO AUTO" %

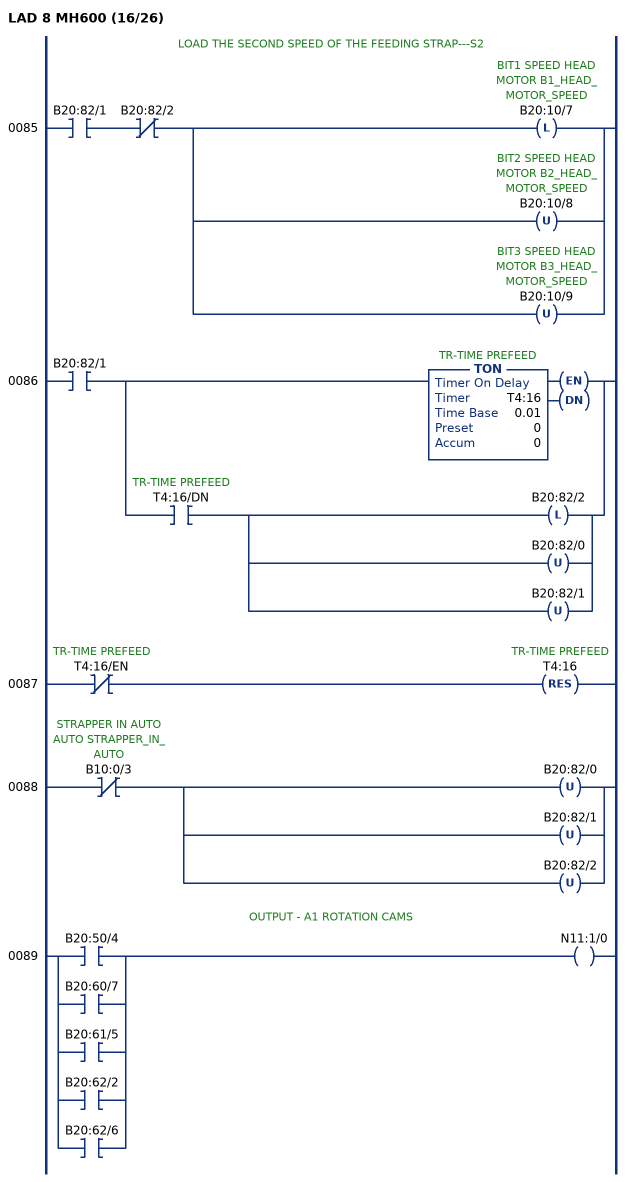
% Rung: 85 %
% LOAD THE SECOND SPEED OF THE FEEDING STRAP---S2 %
SOR XIC B20:82/1 XIO B20:82/2 BST OTL B20:10/7 NXB BST OTU B20:10/8 NXB OTU B20:10/9 BND BND EOR
%   B20:10/7  B1_HEAD_MOTOR_SPEED  "BIT1 SPEED HEAD MOTOR" %
%   B20:10/8  B2_HEAD_MOTOR_SPEED  "BIT2 SPEED HEAD MOTOR" %
%   B20:10/9  B3_HEAD_MOTOR_SPEED  "BIT3 SPEED HEAD MOTOR" %
% Rung: 86 %
SOR XIC B20:82/1 BST TON T4:16 0.01 0 0 NXB XIC T4:16/DN BST OTL B20:82/2 NXB BST OTU B20:82/0 NXB OTU B20:82/1 BND BND BND EOR
%   T4:16  "TR-TIME PREFEED" %
% Rung: 87 %
SOR XIO T4:16/EN RES T4:16 EOR
%   T4:16  "TR-TIME PREFEED" %
% Rung: 88 %
SOR XIO B10:0/3 BST OTU B20:82/0 NXB BST OTU B20:82/1 NXB OTU B20:82/2 BND BND EOR
%   B10:0/3  STRAPPER_IN_AUTO  "STRAPPER IN AUTO AUTO" %
% Rung: 89 %
% OUTPUT - A1 ROTATION CAMS %
SOR BST XIC B20:50/4 NXB BST XIC B20:60/7 NXB BST XIC B20:61/5 NXB BST XIC B20:62/2 NXB XIC B20:62/6 BND BND BND BND OTE N11:1/0 EOR

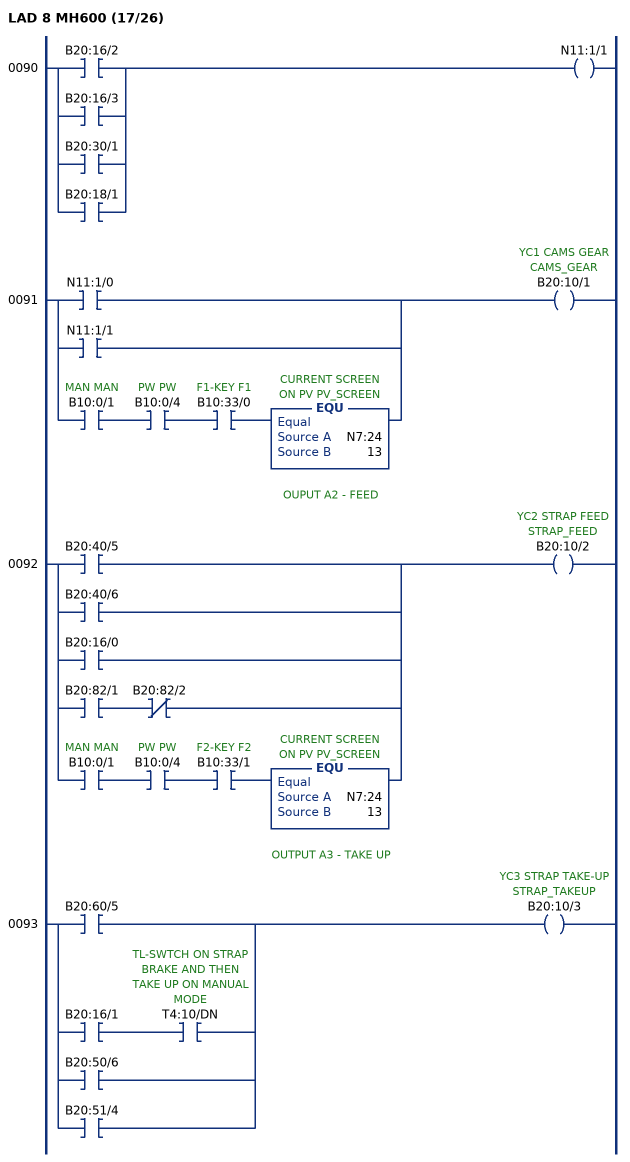
% Rung: 90 %
SOR BST XIC B20:16/2 NXB BST XIC B20:16/3 NXB BST XIC B20:30/1 NXB XIC B20:18/1 BND BND BND OTE N11:1/1 EOR
% Rung: 91 %
SOR BST XIC N11:1/0 NXB BST XIC N11:1/1 NXB XIC B10:0/1 XIC B10:0/4 XIC B10:33/0 EQU N7:24 13 BND BND OTE B20:10/1 EOR
%   B10:0/1  MAN  "MAN" %
%   B10:0/4  PW  "PW" %
%   B10:33/0  F1  "F1-KEY" %
%   N7:24  PV_SCREEN  "CURRENT SCREEN ON PV" %
%   B20:10/1  CAMS_GEAR  "YC1 CAMS GEAR" %
% Rung: 92 %
% OUPUT A2 - FEED %
SOR BST XIC B20:40/5 NXB BST XIC B20:40/6 NXB BST XIC B20:16/0 NXB BST XIC B20:82/1 XIO B20:82/2 NXB XIC B10:0/1 XIC B10:0/4 XIC B10:33/1 EQU N7:24 13 BND BND BND BND OTE B20:10/2 EOR
%   B10:0/1  MAN  "MAN" %
%   B10:0/4  PW  "PW" %
%   B10:33/1  F2  "F2-KEY" %
%   N7:24  PV_SCREEN  "CURRENT SCREEN ON PV" %
%   B20:10/2  STRAP_FEED  "YC2 STRAP FEED" %
% Rung: 93 %
% OUTPUT A3 - TAKE UP %
SOR BST XIC B20:60/5 NXB BST XIC B20:16/1 XIC T4:10/DN NXB BST XIC B20:50/6 NXB XIC B20:51/4 BND BND BND OTE B20:10/3 EOR
%   T4:10  "TL-SWTCH ON STRAP BRAKE AND THEN TAKE UP ON MANUAL MODE" %
%   B20:10/3  STRAP_TAKEUP  "YC3 STRAP TAKE-UP" %

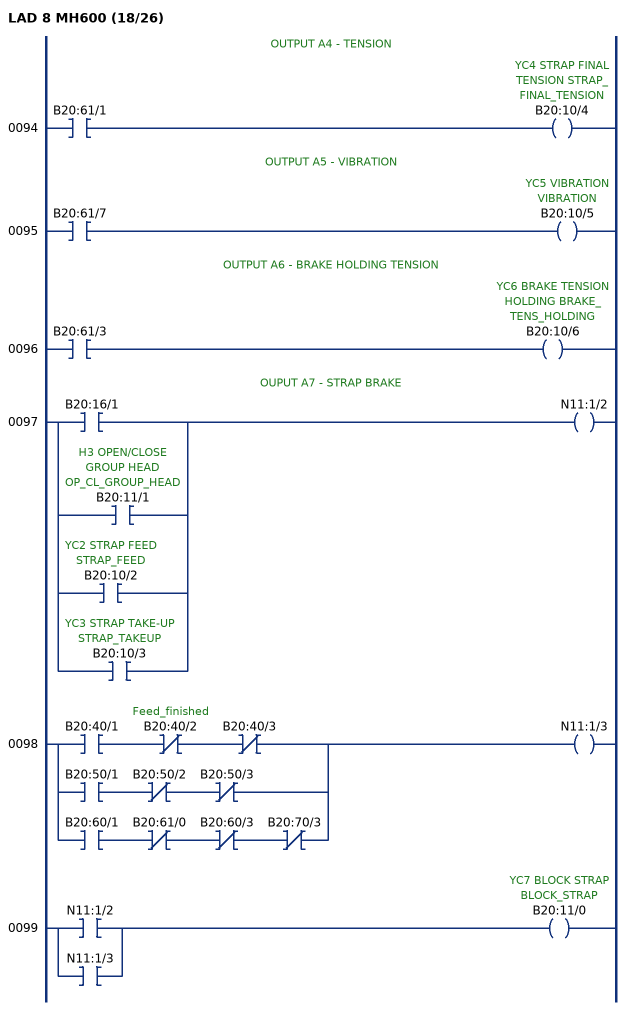
% Rung: 94 %
% OUTPUT A4 - TENSION %
SOR XIC B20:61/1 OTE B20:10/4 EOR
%   B20:10/4  STRAP_FINAL_TENSION  "YC4 STRAP FINAL TENSION" %
% Rung: 95 %
% OUTPUT A5 - VIBRATION %
SOR XIC B20:61/7 OTE B20:10/5 EOR
%   B20:10/5  VIBRATION  "YC5 VIBRATION" %
% Rung: 96 %
% OUTPUT A6 - BRAKE HOLDING TENSION %
SOR XIC B20:61/3 OTE B20:10/6 EOR
%   B20:10/6  BRAKE_TENS_HOLDING  "YC6 BRAKE TENSION HOLDING" %
% Rung: 97 %
% OUPUT A7 - STRAP BRAKE %
SOR BST XIC B20:16/1 NXB BST XIC B20:11/1 NXB BST XIC B20:10/2 NXB XIC B20:10/3 BND BND BND OTE N11:1/2 EOR
%   B20:11/1  OP_CL_GROUP_HEAD  "H3 OPEN/CLOSE GROUP HEAD" %
%   B20:10/2  STRAP_FEED  "YC2 STRAP FEED" %
%   B20:10/3  STRAP_TAKEUP  "YC3 STRAP TAKE-UP" %
% Rung: 98 %
SOR BST XIC B20:40/1 XIO B20:40/2 XIO B20:40/3 NXB BST XIC B20:50/1 XIO B20:50/2 XIO B20:50/3 NXB XIC B20:60/1 XIO B20:61/0 XIO B20:60/3 XIO B20:70/3 BND BND OTE N11:1/3 EOR
%   B20:40/2  "Feed_finished" %
% Rung: 99 %
SOR BST XIC N11:1/2 NXB XIC N11:1/3 BND OTE B20:11/0 EOR
%   B20:11/0  BLOCK_STRAP  "YC7 BLOCK STRAP" %

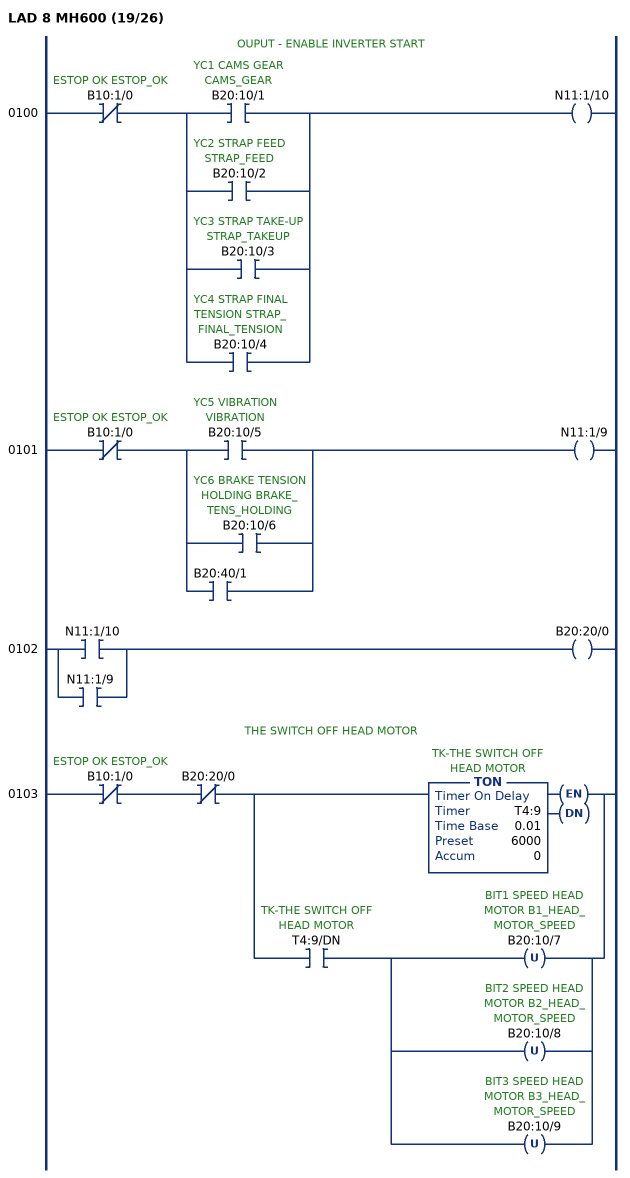
% Rung: 100 %
% OUPUT - ENABLE INVERTER START %
SOR XIO B10:1/0 BST XIC B20:10/1 NXB BST XIC B20:10/2 NXB BST XIC B20:10/3 NXB XIC B20:10/4 BND BND BND OTE N11:1/10 EOR
%   B10:1/0  ESTOP_OK  "ESTOP OK" %
%   B20:10/1  CAMS_GEAR  "YC1 CAMS GEAR" %
%   B20:10/2  STRAP_FEED  "YC2 STRAP FEED" %
%   B20:10/3  STRAP_TAKEUP  "YC3 STRAP TAKE-UP" %
%   B20:10/4  STRAP_FINAL_TENSION  "YC4 STRAP FINAL TENSION" %
% Rung: 101 %
SOR XIO B10:1/0 BST XIC B20:10/5 NXB BST XIC B20:10/6 NXB XIC B20:40/1 BND BND OTE N11:1/9 EOR
%   B10:1/0  ESTOP_OK  "ESTOP OK" %
%   B20:10/5  VIBRATION  "YC5 VIBRATION" %
%   B20:10/6  BRAKE_TENS_HOLDING  "YC6 BRAKE TENSION HOLDING" %
% Rung: 102 %
SOR BST XIC N11:1/10 NXB XIC N11:1/9 BND OTE B20:20/0 EOR
% Rung: 103 %
% THE SWITCH OFF HEAD MOTOR %
SOR XIO B10:1/0 XIO B20:20/0 BST TON T4:9 0.01 6000 0 NXB XIC T4:9/DN BST OTU B20:10/7 NXB BST OTU B20:10/8 NXB OTU B20:10/9 BND BND BND EOR
%   B10:1/0  ESTOP_OK  "ESTOP OK" %
%   T4:9  "TK-THE SWITCH OFF HEAD MOTOR" %
%   B20:10/7  B1_HEAD_MOTOR_SPEED  "BIT1 SPEED HEAD MOTOR" %
%   B20:10/8  B2_HEAD_MOTOR_SPEED  "BIT2 SPEED HEAD MOTOR" %
%   B20:10/9  B3_HEAD_MOTOR_SPEED  "BIT3 SPEED HEAD MOTOR" %

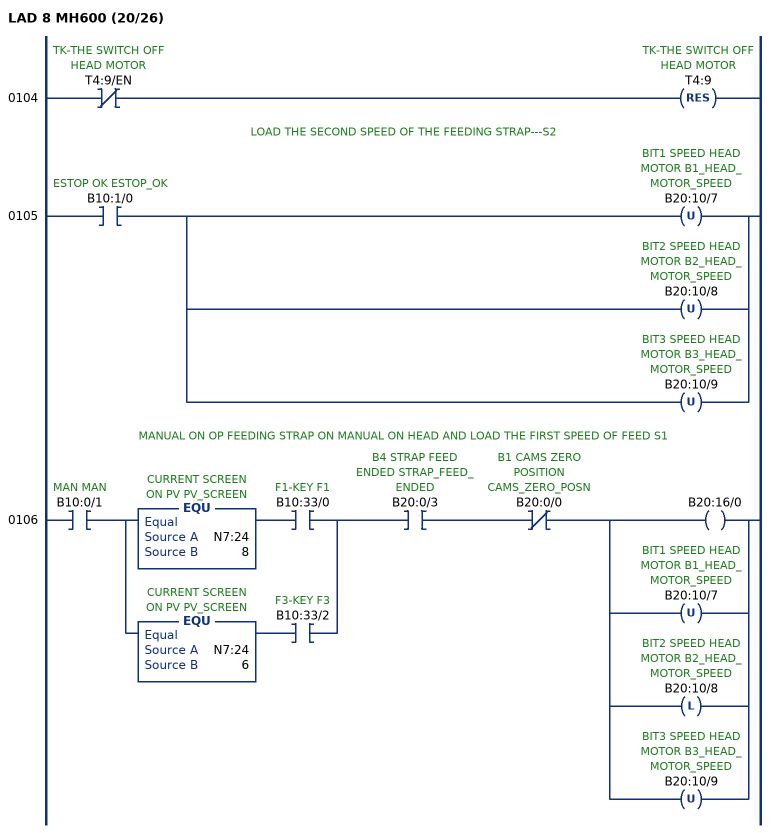
% Rung: 104 %
SOR XIO T4:9/EN RES T4:9 EOR
%   T4:9  "TK-THE SWITCH OFF HEAD MOTOR" %
% Rung: 105 %
% LOAD THE SECOND SPEED OF THE FEEDING STRAP---S2 %
SOR XIC B10:1/0 BST OTU B20:10/7 NXB BST OTU B20:10/8 NXB OTU B20:10/9 BND BND EOR
%   B10:1/0  ESTOP_OK  "ESTOP OK" %
%   B20:10/7  B1_HEAD_MOTOR_SPEED  "BIT1 SPEED HEAD MOTOR" %
%   B20:10/8  B2_HEAD_MOTOR_SPEED  "BIT2 SPEED HEAD MOTOR" %
%   B20:10/9  B3_HEAD_MOTOR_SPEED  "BIT3 SPEED HEAD MOTOR" %
% Rung: 106 %
% MANUAL ON OP FEEDING STRAP ON MANUAL ON HEAD AND LOAD THE FIRST SPEED OF FEED S1 %
SOR XIC B10:0/1 BST EQU N7:24 8 XIC B10:33/0 NXB EQU N7:24 6 XIC B10:33/2 BND XIC B20:0/3 XIO B20:0/0 BST OTE B20:16/0 NXB BST OTU B20:10/7 NXB BST OTL B20:10/8 NXB OTU B20:10/9 BND BND BND EOR
%   B10:0/1  MAN  "MAN" %
%   N7:24  PV_SCREEN  "CURRENT SCREEN ON PV" %
%   B10:33/0  F1  "F1-KEY" %
%   B10:33/2  F3  "F3-KEY" %
%   B20:0/3  STRAP_FEED_ENDED  "B4 STRAP FEED ENDED" %
%   B20:0/0  CAMS_ZERO_POSN  "B1 CAMS ZERO POSITION" %
%   B20:10/7  B1_HEAD_MOTOR_SPEED  "BIT1 SPEED HEAD MOTOR" %
%   B20:10/8  B2_HEAD_MOTOR_SPEED  "BIT2 SPEED HEAD MOTOR" %
%   B20:10/9  B3_HEAD_MOTOR_SPEED  "BIT3 SPEED HEAD MOTOR" %

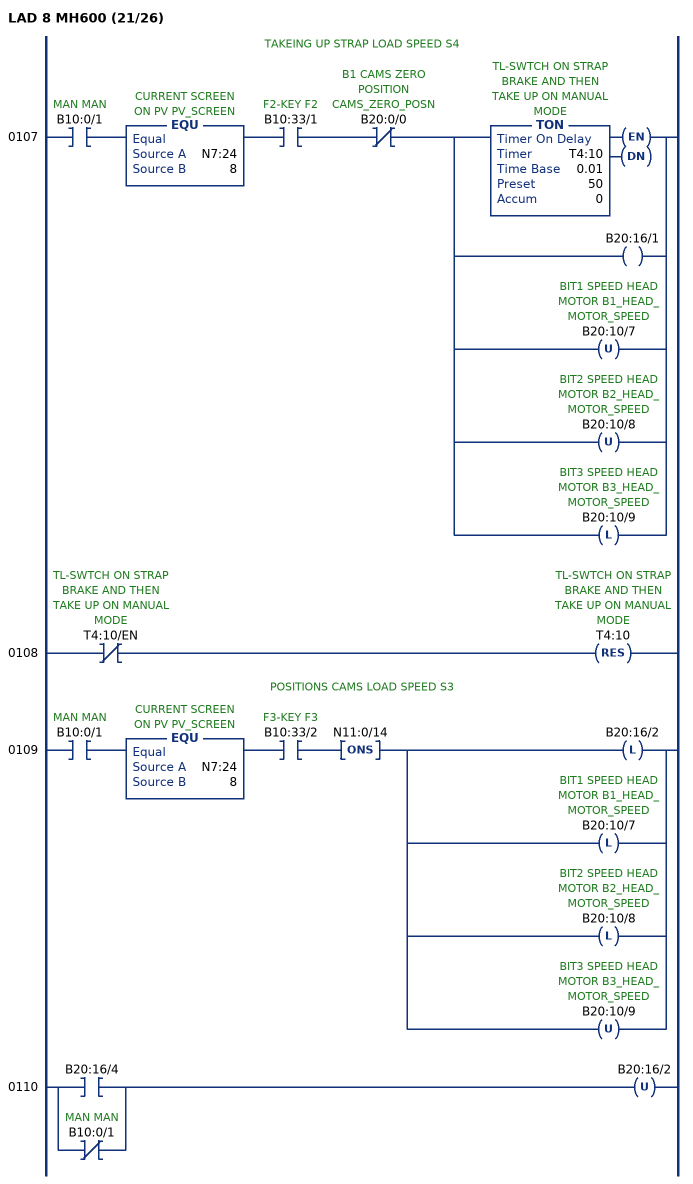
% Rung: 107 %
% TAKEING UP STRAP LOAD SPEED S4 %
SOR XIC B10:0/1 EQU N7:24 8 XIC B10:33/1 XIO B20:0/0 BST TON T4:10 0.01 50 0 NXB BST OTE B20:16/1 NXB BST OTU B20:10/7 NXB BST OTU B20:10/8 NXB OTL B20:10/9 BND BND BND BND EOR
%   B10:0/1  MAN  "MAN" %
%   N7:24  PV_SCREEN  "CURRENT SCREEN ON PV" %
%   B10:33/1  F2  "F2-KEY" %
%   B20:0/0  CAMS_ZERO_POSN  "B1 CAMS ZERO POSITION" %
%   T4:10  "TL-SWTCH ON STRAP BRAKE AND THEN TAKE UP ON MANUAL MODE" %
%   B20:10/7  B1_HEAD_MOTOR_SPEED  "BIT1 SPEED HEAD MOTOR" %
%   B20:10/8  B2_HEAD_MOTOR_SPEED  "BIT2 SPEED HEAD MOTOR" %
%   B20:10/9  B3_HEAD_MOTOR_SPEED  "BIT3 SPEED HEAD MOTOR" %
% Rung: 108 %
SOR XIO T4:10/EN RES T4:10 EOR
%   T4:10  "TL-SWTCH ON STRAP BRAKE AND THEN TAKE UP ON MANUAL MODE" %
% Rung: 109 %
% POSITIONS CAMS LOAD SPEED S3 %
SOR XIC B10:0/1 EQU N7:24 8 XIC B10:33/2 ONS N11:0/14 BST OTL B20:16/2 NXB BST OTL B20:10/7 NXB BST OTL B20:10/8 NXB OTU B20:10/9 BND BND BND EOR
%   B10:0/1  MAN  "MAN" %
%   N7:24  PV_SCREEN  "CURRENT SCREEN ON PV" %
%   B10:33/2  F3  "F3-KEY" %
%   B20:10/7  B1_HEAD_MOTOR_SPEED  "BIT1 SPEED HEAD MOTOR" %
%   B20:10/8  B2_HEAD_MOTOR_SPEED  "BIT2 SPEED HEAD MOTOR" %
%   B20:10/9  B3_HEAD_MOTOR_SPEED  "BIT3 SPEED HEAD MOTOR" %
% Rung: 110 %
SOR BST XIC B20:16/4 NXB XIO B10:0/1 BND OTU B20:16/2 EOR
%   B10:0/1  MAN  "MAN" %

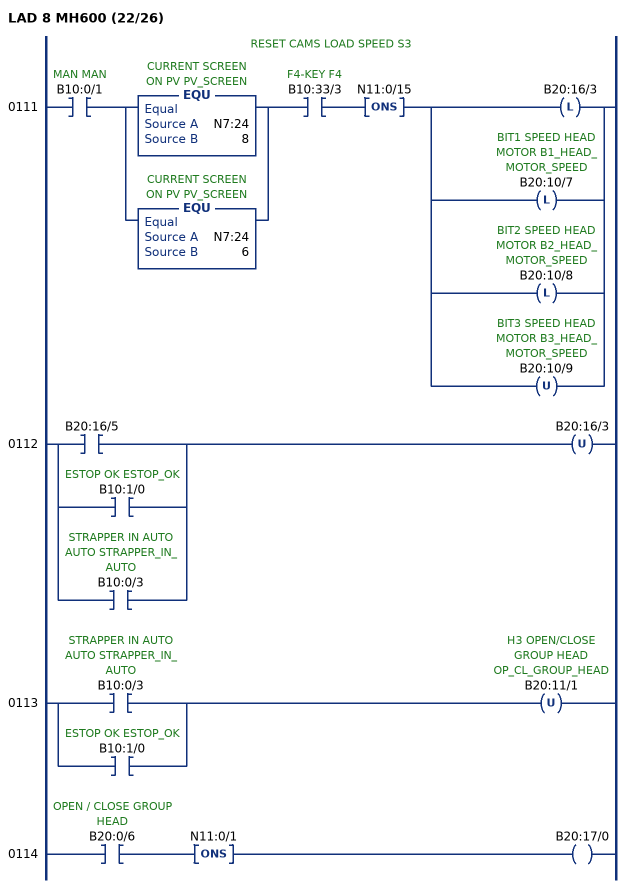
% Rung: 111 %
% RESET CAMS LOAD SPEED S3 %
SOR XIC B10:0/1 BST EQU N7:24 8 NXB EQU N7:24 6 BND XIC B10:33/3 ONS N11:0/15 BST OTL B20:16/3 NXB BST OTL B20:10/7 NXB BST OTL B20:10/8 NXB OTU B20:10/9 BND BND BND EOR
%   B10:0/1  MAN  "MAN" %
%   N7:24  PV_SCREEN  "CURRENT SCREEN ON PV" %
%   B10:33/3  F4  "F4-KEY" %
%   B20:10/7  B1_HEAD_MOTOR_SPEED  "BIT1 SPEED HEAD MOTOR" %
%   B20:10/8  B2_HEAD_MOTOR_SPEED  "BIT2 SPEED HEAD MOTOR" %
%   B20:10/9  B3_HEAD_MOTOR_SPEED  "BIT3 SPEED HEAD MOTOR" %
% Rung: 112 %
SOR BST XIC B20:16/5 NXB BST XIC B10:1/0 NXB XIC B10:0/3 BND BND OTU B20:16/3 EOR
%   B10:1/0  ESTOP_OK  "ESTOP OK" %
%   B10:0/3  STRAPPER_IN_AUTO  "STRAPPER IN AUTO AUTO" %
% Rung: 113 %
SOR BST XIC B10:0/3 NXB XIC B10:1/0 BND OTU B20:11/1 EOR
%   B10:0/3  STRAPPER_IN_AUTO  "STRAPPER IN AUTO AUTO" %
%   B10:1/0  ESTOP_OK  "ESTOP OK" %
%   B20:11/1  OP_CL_GROUP_HEAD  "H3 OPEN/CLOSE GROUP HEAD" %
% Rung: 114 %
SOR XIC B20:0/6 ONS N11:0/1 OTE B20:17/0 EOR
%   B20:0/6  "OPEN / CLOSE GROUP HEAD" %

